# EPICS substitutions: iocBoot/iocZed/zedLOreg0.substitutions
file "$(TOP)/zzzApp/Db/zedLOreg.template"
{
pattern
{P,R,C,N}
{zzz:,reg0_,0,0}
{zzz:,reg0_,0,1}
{zzz:,reg0_,0,2}
{zzz:,reg0_,0,3}
{zzz:,reg0_,0,4}
{zzz:,reg0_,0,5}
{zzz:,reg0_,0,6}
{zzz:,reg0_,0,7}
{zzz:,reg0_,0,8}
{zzz:,reg0_,0,9}
{zzz:,reg0_,0,10}
{zzz:,reg0_,0,11}
{zzz:,reg0_,0,12}
{zzz:,reg0_,0,13}
{zzz:,reg0_,0,14}
{zzz:,reg0_,0,15}
{zzz:,reg0_,0,16}
{zzz:,reg0_,0,17}
{zzz:,reg0_,0,18}
{zzz:,reg0_,0,19}
{zzz:,reg0_,0,20}
{zzz:,reg0_,0,21}
{zzz:,reg0_,0,22}
{zzz:,reg0_,0,23}
{zzz:,reg0_,0,24}
{zzz:,reg0_,0,25}
{zzz:,reg0_,0,26}
{zzz:,reg0_,0,27}
{zzz:,reg0_,0,28}
{zzz:,reg0_,0,29}

{zzz:,reg0_,0,30}
{zzz:,reg0_,0,31}
{zzz:,reg0_,0,32}
{zzz:,reg0_,0,33}
{zzz:,reg0_,0,34}
{zzz:,reg0_,0,35}
{zzz:,reg0_,0,36}
{zzz:,reg0_,0,37}
{zzz:,reg0_,0,38}
{zzz:,reg0_,0,39}

{zzz:,reg0_,0,40}
{zzz:,reg0_,0,41}
{zzz:,reg0_,0,42}
{zzz:,reg0_,0,43}
{zzz:,reg0_,0,44}
{zzz:,reg0_,0,45}
{zzz:,reg0_,0,46}
{zzz:,reg0_,0,47}
{zzz:,reg0_,0,48}
{zzz:,reg0_,0,49}

{zzz:,reg0_,0,50}
{zzz:,reg0_,0,51}
{zzz:,reg0_,0,52}
{zzz:,reg0_,0,53}
{zzz:,reg0_,0,54}
{zzz:,reg0_,0,55}
{zzz:,reg0_,0,56}
{zzz:,reg0_,0,57}
{zzz:,reg0_,0,58}
{zzz:,reg0_,0,59}

{zzz:,reg0_,0,60}
{zzz:,reg0_,0,61}
{zzz:,reg0_,0,62}
{zzz:,reg0_,0,63}
{zzz:,reg0_,0,64}
{zzz:,reg0_,0,65}
{zzz:,reg0_,0,66}
{zzz:,reg0_,0,67}
{zzz:,reg0_,0,68}
{zzz:,reg0_,0,69}

{zzz:,reg0_,0,70}
{zzz:,reg0_,0,71}
{zzz:,reg0_,0,72}
{zzz:,reg0_,0,73}
{zzz:,reg0_,0,74}
{zzz:,reg0_,0,75}
{zzz:,reg0_,0,76}
{zzz:,reg0_,0,77}
{zzz:,reg0_,0,78}
{zzz:,reg0_,0,79}

{zzz:,reg0_,0,80}
{zzz:,reg0_,0,81}
{zzz:,reg0_,0,82}
{zzz:,reg0_,0,83}
{zzz:,reg0_,0,84}
{zzz:,reg0_,0,85}
{zzz:,reg0_,0,86}
{zzz:,reg0_,0,87}
{zzz:,reg0_,0,88}
{zzz:,reg0_,0,89}

{zzz:,reg0_,0,90}
{zzz:,reg0_,0,91}
{zzz:,reg0_,0,92}
{zzz:,reg0_,0,93}
{zzz:,reg0_,0,94}
{zzz:,reg0_,0,95}
{zzz:,reg0_,0,96}
{zzz:,reg0_,0,97}
{zzz:,reg0_,0,98}
{zzz:,reg0_,0,99}

{zzz:,reg0_,0,100}
{zzz:,reg0_,0,101}
{zzz:,reg0_,0,102}
{zzz:,reg0_,0,103}
{zzz:,reg0_,0,104}
{zzz:,reg0_,0,105}
{zzz:,reg0_,0,106}
{zzz:,reg0_,0,107}
{zzz:,reg0_,0,108}
{zzz:,reg0_,0,109}

{zzz:,reg0_,0,110}
{zzz:,reg0_,0,111}
{zzz:,reg0_,0,112}
{zzz:,reg0_,0,113}
{zzz:,reg0_,0,114}
{zzz:,reg0_,0,115}
{zzz:,reg0_,0,116}
{zzz:,reg0_,0,117}
{zzz:,reg0_,0,118}
{zzz:,reg0_,0,119}

{zzz:,reg0_,0,120}
{zzz:,reg0_,0,121}
{zzz:,reg0_,0,122}
{zzz:,reg0_,0,123}
{zzz:,reg0_,0,124}
{zzz:,reg0_,0,125}
{zzz:,reg0_,0,126}
{zzz:,reg0_,0,127}
{zzz:,reg0_,0,128}
{zzz:,reg0_,0,129}

{zzz:,reg0_,0,130}
{zzz:,reg0_,0,131}
{zzz:,reg0_,0,132}
{zzz:,reg0_,0,133}
{zzz:,reg0_,0,134}
{zzz:,reg0_,0,135}
{zzz:,reg0_,0,136}
{zzz:,reg0_,0,137}
{zzz:,reg0_,0,138}
{zzz:,reg0_,0,139}
}
